TYPE tstCTCProcessDataIn :
STRUCT
	State			:USINT;		
	stStatusBits	:tstCTCStatusBits;	
	ActualForce 	:REAL;		
	ActualSpeed 	:REAL;		
	ActualPosition 	:REAL;		
END_STRUCT
END_TYPE

(* stored: Version 1.1.0.1, ProductVersion 3.1.4026.17
   DUT tstCTCProcessDataIn: Id {5038f597-1a64-4609-9c55-3d8d86ca2731} *)
